{attribute 'GeneratedUsingTerminal: EP1122-0001-0018'}
{attribute addProperty BoxType "EP1122-0001-0018"}
{attribute addProperty Id "A_0027_EP1258_0001_0016EP1258_7DB9B57056A_0028_EP1258_0001_0017EP1258_7DB9B57056A_0029_EP1258_0001_0018EP1258_7DB9B57056A_0030_EP1258_0001_0019EP1258_7DB9B57056A_0031_EP1258_0001_0020EP1258_7DB9B57056A_0032_EP1258_0002_0016EP1258_7DB9B57056A_0033_EP1258_0002_0017EP1258_7DB9B57056A_0034_EP1258_0002_0018EP1258_7DB9B57056A_0035_EP1258_0002_0019EP1258_7DB9B57056A_0036_EP1258_0002_0020EP1258_7DB9B57056A_0037_EP1312_0001_0016A_0037_EP1312_0001_0016_A4C0FB61890"}
{attribute addProperty CRC "3845022899"}
{attribute addProperty Size "1450"}
TYPE A_0026_EP1122_0001_0018_E52E64B3 EXTENDS EP1122_AB5A9467 :
STRUCT
	{attribute addProperty Name "A_0027_EP1258_0001_0016"}
	A_0027_EP1258_0001_0016 : EP1258_7DB9B570;
	{attribute addProperty Name "A_0028_EP1258_0001_0017"}
	A_0028_EP1258_0001_0017 : EP1258_7DB9B570;
	{attribute addProperty Name "A_0029_EP1258_0001_0018"}
	A_0029_EP1258_0001_0018 : EP1258_7DB9B570;
	{attribute addProperty Name "A_0030_EP1258_0001_0019"}
	A_0030_EP1258_0001_0019 : EP1258_7DB9B570;
	{attribute addProperty Name "A_0031_EP1258_0001_0020"}
	A_0031_EP1258_0001_0020 : EP1258_7DB9B570;
	{attribute addProperty Name "A_0032_EP1258_0002_0016"}
	A_0032_EP1258_0002_0016 : EP1258_7DB9B570;
	{attribute addProperty Name "A_0033_EP1258_0002_0017"}
	A_0033_EP1258_0002_0017 : EP1258_7DB9B570;
	{attribute addProperty Name "A_0034_EP1258_0002_0018"}
	A_0034_EP1258_0002_0018 : EP1258_7DB9B570;
	{attribute addProperty Name "A_0035_EP1258_0002_0019"}
	A_0035_EP1258_0002_0019 : EP1258_7DB9B570;
	{attribute addProperty Name "A_0036_EP1258_0002_0020"}
	A_0036_EP1258_0002_0020 : EP1258_7DB9B570;
	{attribute addProperty Name "A_0037_EP1312_0001_0016"}
	A_0037_EP1312_0001_0016 : A_0037_EP1312_0001_0016_A4C0FB61;
END_STRUCT
END_TYPE

(* stored: Version 1.2.0.0, ProductVersion 3.1.4024.9
   DUT A_0026_EP1122_0001_0018_E52E64B3: Id {48e50c52-1573-4c94-8d39-410125091a9c} *)
